SUBAPPLICATION GreenWhiteBackground1_AX (* Hintergrundfarbe (TRUE -> Grün, FALSE -> Weiß) für 1 Objekt (AX-Adapter) *)
  (* Standard: 61499-2; Description: Copyright (c) 2022 HR Agrartechnik GmbH This program and the accompanying materials are made available under the terms of the Eclipse Public License 2.0 which is available at https://www.eclipse.org/legal/epl-2.0/ SPDX-License-Identifier: EPL-2.0 *)
  (* Version 1.0, 2022-11-10, Franz Höpfinger, HR Agrartechnik GmbH *)
  PACKAGE MyLib::sys;
  IMPORT isobus::UT::Q::const::IDs::ID_NULL;
  IMPORT isobus::UT::Q::const::colours::COLOR_GREEN;
  IMPORT isobus::UT::Q::const::colours::COLOR_WHITE;
  (* Documentation:
  Hintergrundfarbe für ein normales VT-Objekt
   Setzt die Hintergrundfarbe (TRUE -> Grün, FALSE -> Weiß) eines einzelnen normalen VT-Objekts (SoftKey, Button, Output-Feld, Container usw.) über u16ObjId. Sendet dafür genau ein ISO-11783-6-Kommando (Part 6 - F.20, "Change Background Colour", FB Q_BackgroundColour) an das VT.
   Für ein Auxiliary-Function-Type-2-Objekt (Object-ID-Bereich 31000–31999) reicht dieser Baustein nicht, weil dessen Zuweisung zusätzlich am physischen Aux-Handle (Joystick) angezeigt wird und dafür ein zweites Kommando über die Aux-Verbindung nötig ist - dafür GreenWhiteBackground2_AX verwenden. Für die Kombination "1 normales Objekt + 1 Aux-Objekt gemeinsam schalten" GreenWhiteBackground3_AX verwenden.
  *)
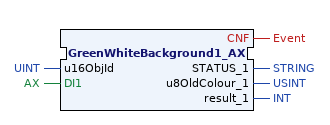
  EVENT_OUTPUT
    CNF; (* Execution Confirmation *)
  END_EVENT
  VAR_INPUT
    u16ObjId : UINT := ID_NULL; (* Object ID Softkey/Button *)
  END_VAR
  VAR_OUTPUT
    STATUS_1 : STRING; (* Service Status *)
    u8OldColour_1 : USINT; (* Old value of ID *)
    result_1 : INT; (* retval see description *)
  END_VAR
  SOCKETS
    DI1 : adapter::types::unidirectional::AX; (* Selector *)
  END_SOCKETS
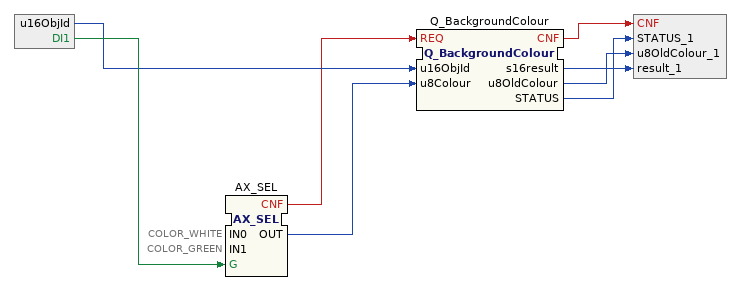
  FBS
    Q_BackgroundColour : isobus::UT::Q::Q_BackgroundColour;
    AX_SEL : adapter::iec61131::selection::AX_SEL(IN0 := COLOR_WHITE, IN1 := COLOR_GREEN);
  END_FBS
  EVENT_CONNECTIONS
    Q_BackgroundColour.CNF TO CNF;
    AX_SEL.CNF TO Q_BackgroundColour.REQ;
  END_CONNECTIONS
  DATA_CONNECTIONS
    u16ObjId TO Q_BackgroundColour.u16ObjId;
    Q_BackgroundColour.s16result TO result_1;
    Q_BackgroundColour.u8OldColour TO u8OldColour_1;
    Q_BackgroundColour.STATUS TO STATUS_1;
    AX_SEL.OUT TO Q_BackgroundColour.u8Colour;
  END_CONNECTIONS
  ADAPTER_CONNECTIONS
    DI1 TO AX_SEL.G;
  END_CONNECTIONS
END_SUBAPPLICATION
